{attribute 'GeneratedUsingTerminal: KL6211-0002'}
{attribute addProperty BoxType "KL6211-0002"}
{attribute addProperty Id "Channel_1AT %Q*Channel_82ADD0760"}
{attribute addProperty CRC "4227989944"}
{attribute addProperty Size "0"}
TYPE KL_FC0201B8 :
STRUCT
	{attribute addProperty Name "Channel_1"}
	Channel_1 : Channel_82ADD076;
END_STRUCT
END_TYPE

(* stored: Version 1.2.0.0, ProductVersion 3.1.4024.9
   DUT KL_FC0201B8: Id {4586cf3a-b2e4-4bae-a80e-8d5df76c9d18} *)
